DATA_BLOCK "ID_PE_Plate_Measure"
{ S7_Optimized_Access := 'TRUE' }
VERSION : 0.1
NON_RETAIN
"FB_PE_Plate_Measure"

BEGIN

END_DATA_BLOCK

